// TIA Portal V19 export
FUNCTION_BLOCK "FB_QF"   // FB31, LAD
TITLE = Querförderer
{ S7_Optimized_Access := 'TRUE' }
// stored: AutoNumber false, MemoryReserve 100, SetENOAutomatically true
   VAR RETAIN
      In { ExternalAccessible := 'False'; ExternalVisible := 'False'; ExternalWritable := 'False'} : Struct
         NotHalt : Bool;
         Auto : Bool;
         Hand : Bool;
         Tipp : Bool;
         T_WR02_zu_UE : Bool;
         T_WR02_zu_BE : Bool;
         T_WR03_zu_UE : Bool;
         T_WR03_zu_BE : Bool;
         S_WR02_lgsm_UE : Bool;
         S_WR02_lgsm_BE : Bool;
         S_WR03_lgsm_UE : Bool;
         S_WR03_lgsm_BE : Bool;
         S_WR02_UE : Bool;
         S_WR02_BE : Bool;
         S_WR03_UE : Bool;
         S_WR03_BE : Bool;
         Req_Ausfahrt_GO : Bool;
         Req_Aufgabe_GO : Bool;
         FU_betriebsbereit_WR02 : Bool;
         FU_betriebsbereit_WR03 : Bool;
         FU_Stoerung_WR02 : Bool;
         FU_Stoerung_WR03 : Bool;
         ErrQ : Bool;
         FU_speed_WR02 : Int;
         FU_speed_WR03 : Int;
      END_STRUCT;
      Param { ExternalAccessible := 'False'; ExternalVisible := 'False'; ExternalWritable := 'False'} : Struct
         "TO" : Time := T#48s;
      END_STRUCT;
      Zst { ExternalAccessible := 'False'; ExternalVisible := 'False'; ExternalWritable := 'False'} : Struct
         Fehler : Bool;
         Req_WR02_In : Bool;
         Req_WR03_In : Bool;
         Req_WR02_Out : Bool;
         Req_WR03_Out : Bool;
         Tor_sicher : Bool;
         TW_sicher : Bool;
      END_STRUCT;
      Out { ExternalAccessible := 'False'; ExternalVisible := 'False'; ExternalWritable := 'False'} : Struct
         WR02_einfahren : Bool;   // zur ÜbergabeStation
         WR02_ausfahren : Bool;   // zum Be-/Entladen
         WR03_einfahren : Bool;   // zur ÜbergabeStation
         WR03_ausfahren : Bool;   // zum Be-/Entladen
         Soll_speed_WR02 : Int;
         Soll_speed_WR03 : Int;
      END_STRUCT;
      Mld { ExternalAccessible := 'False'; ExternalVisible := 'False'; ExternalWritable := 'False'} : Struct
         TO_WR02 : Bool;
         TO_WR03 : Bool;
         St_FU_WR02 : Bool;
         St_FU_WR03 : Bool;
         FU_nichtbereit_WR02 : Bool;
         FU_nichtbereit_WR03 : Bool;
         n_Auto : Bool;
         SF_WR02 : Bool;
         SF_WR03 : Bool;
      END_STRUCT;
   END_VAR
   VAR
      IEC_Timer { ExternalAccessible := 'False'; ExternalVisible := 'False'; ExternalWritable := 'False'} : Struct
         TO_WR02 { S7_SetPoint := 'True'} : TON_TIME;
         TO_WR03 { S7_SetPoint := 'True'} : TON_TIME;
      END_STRUCT;
   END_VAR
   VAR_TEMP
      TO_WR02 : Bool;
      TO_WR03 : Bool;
   END_VAR
   VAR CONSTANT
      Speed_Tipp : Int := 25;   // %
      Speed_Hand : Int := 70;   // %
      Speed_Auto : Int := 70;   // % == 35 Hz = 150 mm/s
   END_VAR
BEGIN

REGION Network 1 (SCL): Input
   // Panelbedienung und Sensoren --> Input()
   // Not-Halt
   #In.NotHalt := NOT "DB_PNOZ_IN_Out".In.NH_Frg_TW_QF;
   // Rolltor
   #Zst.Tor_sicher := "Tor".In.S_auf AND NOT "Tor".Out.zu;
   // Transportwagen 
   #Zst.TW_sicher := "DI_FW_1".ZST.PosInc < ("DB_POS".POS[25].IncPos - "DB_POS".POS[25].IncAbstand_rck);

   // Anforderung Automatikbetrieb
   IF #In.Auto THEN
       "FC_Anf_BE"(Req_GO_Ausfahrt := #In.Req_Ausfahrt_GO,
                   Req_GO_Aufgabe := #In.Req_Aufgabe_GO,
                   Req_WR02_IN := #Zst.Req_WR02_In,
                   Req_WR02_OUT := #Zst.Req_WR02_Out,
                   Req_WR03_IN := #Zst.Req_WR03_In,
                   Req_WR03_OUT := #Zst.Req_WR03_Out);
   ELSE
       #Zst.Req_WR02_In := FALSE;
       #Zst.Req_WR02_Out := FALSE;
       #Zst.Req_WR03_In := FALSE;
       #Zst.Req_WR03_Out := FALSE;
   END_IF;
END_REGION

REGION Network 2 (SCL): Sammelstörung
   IF #In.ErrQ THEN
       #Zst.Fehler := FALSE;
   END_IF;

   IF #In.NotHalt OR #Mld.FU_nichtbereit_WR02 OR #Mld.FU_nichtbereit_WR03 OR #Mld.SF_WR02
       OR #Mld.SF_WR03 OR #Mld.St_FU_WR02 OR #Mld.St_FU_WR03 OR #Mld.TO_WR02 OR #Mld.TO_WR03  THEN
       #Zst.Fehler := TRUE;
   END_IF;
END_REGION

REGION Network 3 (SCL): Ansteuerung
   IF NOT #Zst.Fehler AND #Zst.Tor_sicher AND #Zst.TW_sicher THEN
       IF #In.Auto THEN // Automatikbetrieb
           // WR02
           #Out.WR02_einfahren := #Zst.Req_WR02_In;
           #Out.WR02_ausfahren := #Zst.Req_WR02_Out;
           // WR03
           #Out.WR03_einfahren := #Zst.Req_WR03_In;
           #Out.WR03_ausfahren := #Zst.Req_WR03_Out;

       ELSIF #In.Hand THEN // Handbetrieb

           // WR02
           IF #In.T_WR02_zu_UE AND NOT #In.T_WR02_zu_BE THEN
               #Out.WR02_einfahren := TRUE;
               #Out.WR02_ausfahren := FALSE;
           END_IF;
           IF #In.T_WR02_zu_BE AND NOT #In.T_WR02_zu_UE THEN
               #Out.WR02_ausfahren := TRUE;
               #Out.WR02_einfahren := FALSE;
           END_IF;
           // WR03
           IF #In.T_WR03_zu_UE AND NOT #In.T_WR03_zu_BE THEN
               #Out.WR03_einfahren := TRUE;
               #Out.WR03_ausfahren := FALSE;
           END_IF;
           IF #In.T_WR03_zu_BE AND NOT #In.T_WR03_zu_UE THEN
               #Out.WR03_ausfahren := TRUE;
               #Out.WR03_einfahren := FALSE;
           END_IF;
       ELSIF #In.Tipp THEN  // Tippbetrieb
           // WR02
           #Out.WR02_einfahren := #In.T_WR02_zu_UE AND NOT #In.T_WR02_zu_BE;
           #Out.WR02_ausfahren := #In.T_WR02_zu_BE AND NOT #In.T_WR02_zu_UE;

           // WR03
           #Out.WR03_einfahren := #In.T_WR03_zu_UE AND NOT #In.T_WR03_zu_BE;
           #Out.WR03_ausfahren := #In.T_WR03_zu_BE AND NOT #In.T_WR03_zu_UE;
       ELSE
           #Out.WR02_einfahren := FALSE;
           #Out.WR02_ausfahren := FALSE;
           #Out.WR03_einfahren := FALSE;
           #Out.WR03_ausfahren := FALSE;

       END_IF;

   ELSE // Not-Halt
       #Out.WR02_einfahren := FALSE;
       #Out.WR02_ausfahren := FALSE;
       #Out.WR03_einfahren := FALSE;
       #Out.WR03_ausfahren := FALSE;

   END_IF;

   // Endlagen erreicht
   IF #In.S_WR02_UE THEN
       #Out.WR02_einfahren := FALSE;
       #Zst.Req_WR02_In := FALSE;
   END_IF;
   IF #In.S_WR02_BE THEN
       #Out.WR02_ausfahren := FALSE;
       #Zst.Req_WR02_Out := FALSE;
   END_IF;
   IF #In.S_WR03_UE THEN
       #Out.WR03_einfahren := FALSE;
       #Zst.Req_WR03_In := FALSE;
   END_IF;
   IF #In.S_WR03_BE THEN
       #Out.WR03_ausfahren := FALSE;
       #Zst.Req_WR03_Out := FALSE;
   END_IF;

   // Geschwindigkeitsvorgabe WR02
   IF NOT #Out.WR02_einfahren AND NOT #Out.WR02_ausfahren THEN
       #Out.Soll_speed_WR02 := 0;
   ELSIF #In.Tipp THEN
       #Out.Soll_speed_WR02 := #Speed_Tipp;
   ELSIF #In.Hand THEN
       #Out.Soll_speed_WR02 := #Speed_Hand;
   ELSE
       #Out.Soll_speed_WR02 := #Speed_Auto;
   END_IF;
   // Positionierung
   IF (#Out.WR02_einfahren AND #In.S_WR02_lgsm_UE) OR (#Out.WR02_ausfahren AND #In.S_WR02_lgsm_BE)THEN
       #Out.Soll_speed_WR02 := #Speed_Tipp;
   END_IF;

   // Geschwindigkeitsvorgabe WR03
   IF NOT #Out.WR03_einfahren AND NOT #Out.WR03_ausfahren THEN
       #Out.Soll_speed_WR03 := 0;
   ELSIF #In.Tipp THEN
       #Out.Soll_speed_WR03 := #Speed_Tipp;
   ELSIF #In.Hand THEN
       #Out.Soll_speed_WR03 := #Speed_Hand;
   ELSE
       #Out.Soll_speed_WR03 := #Speed_Auto;
   END_IF;
   // Positionierung
   IF (#Out.WR03_einfahren AND #In.S_WR03_lgsm_UE) OR (#Out.WR03_ausfahren AND #In.S_WR03_lgsm_BE) THEN
       #Out.Soll_speed_WR03 := #Speed_Tipp;
   END_IF;
END_REGION

REGION Network 4 (SCL): Überwachung / Alarme
   // Störung FU WR02
   #Mld.St_FU_WR02 := #In.FU_Stoerung_WR02 AND NOT #In.NotHalt;
   // Störung FU WR03
   #Mld.St_FU_WR03 := #In.FU_Stoerung_WR03 AND NOT #In.NotHalt;
   // 24V-Betrieb
   #Mld.FU_nichtbereit_WR02 := NOT #In.FU_betriebsbereit_WR02 AND NOT #In.NotHalt;
   #Mld.FU_nichtbereit_WR03 := NOT #In.FU_betriebsbereit_WR03 AND NOT #In.NotHalt;

   // nicht in Automatik
   #Mld.n_Auto := NOT #In.Auto AND "DB_ANLAGE".BA.Automat_ein;

   // Zeitüberschreitung WR02
   #IEC_Timer.TO_WR02(IN := (#Out.WR02_einfahren AND NOT #In.S_WR02_UE) OR (#Out.WR02_ausfahren AND NOT #In.S_WR02_BE),
                        PT := #Param.TO,
                        Q => #TO_WR02);
     IF #TO_WR02 AND #In.Auto THEN
         #Mld.TO_WR02 := TRUE;
     ELSIF #In.ErrQ THEN
         #Mld.TO_WR02 := FALSE;
     END_IF;
   // Zeitüberschreitung WR03
     #IEC_Timer.TO_WR02(IN := (#Out.WR03_einfahren AND NOT #In.S_WR03_UE) OR (#Out.WR03_ausfahren AND NOT #In.S_WR03_BE),
                        PT := #Param.TO,
                        Q => #TO_WR03);
     IF #TO_WR03 AND #In.Auto THEN
         #Mld.TO_WR03 := TRUE;
     ELSIF #In.ErrQ THEN
         #Mld.TO_WR03 := FALSE;
     END_IF;
     //Sensorfehler
     #Mld.SF_WR02 := #In.S_WR02_UE AND #In.S_WR02_BE;
     #Mld.SF_WR03 := #In.S_WR03_UE AND #In.S_WR03_BE;
END_REGION
END_FUNCTION_BLOCK
